FUNCTION_BLOCK TaskCenterMSGParse (* Service Interface Function Block Type *)
  (* Standard: 61499-2 *)
  (* Version 0.0, 2018-06-21, 4DIAC-IDE, 4DIAC-Consortium *)
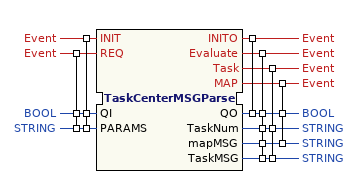
  EVENT_INPUT
    INIT WITH QI, PARAMS; (* Service Initialization *)
    REQ WITH QI, PARAMS; (* Service Request *)
  END_EVENT
  EVENT_OUTPUT
    INITO WITH QO; (* Initialization Confirm *)
    Evaluate WITH QO, TaskMSG, TaskNum, mapMSG; (* Indication from Resource *)
    Task WITH TaskMSG, TaskNum;
    MAP WITH QO, mapMSG;
  END_EVENT
  VAR_INPUT
    QI : BOOL; (* Event Input Qualifier *)
    PARAMS : STRING; (* Service Parameters *)
  END_VAR
  VAR_OUTPUT
    QO : BOOL; (* Event Output Qualifier *)
    TaskNum : STRING;
    mapMSG : STRING; (* MAP msg *)
    TaskMSG : STRING; (* Input data from resource *)
  END_VAR
  SERVICE APPLICATION/RESOURCE (* Service Interface Function Block Type *)
    SEQUENCE normal_establishment
      APPLICATION.INIT+(PARAMS) -> RESOURCE.initialize(PARAMS) -> APPLICATION.INITO+();
    END_SEQUENCE
    SEQUENCE unsuccessful_establishment
      APPLICATION.INIT+(PARAMS) -> RESOURCE.initialize(PARAMS) -> APPLICATION.INITO-(STATUS);
    END_SEQUENCE
    SEQUENCE request_confirm
      APPLICATION.REQ+(SD) -> RESOURCE.request(SD) -> APPLICATION.CNF+(RD);
    END_SEQUENCE
    SEQUENCE request_inhibited
      APPLICATION.REQ-(SD) -> APPLICATION.CNF-(STATUS);
    END_SEQUENCE
    SEQUENCE request_error
      APPLICATION.REQ+(SD) -> RESOURCE.request(SD) -> APPLICATION.CNF-(STATUS);
    END_SEQUENCE
    SEQUENCE indication_response
      RESOURCE.indicate(RD) -> APPLICATION.IND+(RD);
      APPLICATION.RSP(QI,SD) -> RESOURCE.response(QI,SD);
    END_SEQUENCE
    SEQUENCE indication_inhibited
      RESOURCE.indicate(RD,QI=FALSE) -> RESOURCE.inhibited();
    END_SEQUENCE
    SEQUENCE error_indication
      RESOURCE.error(STATUS) -> APPLICATION.IND-(STATUS);
    END_SEQUENCE
    SEQUENCE application_initiated_termination
      APPLICATION.INIT-() -> RESOURCE.terminate() -> APPLICATION.INITO-(STATUS);
    END_SEQUENCE
    SEQUENCE resource_initiated_termination
      -> APPLICATION.INITO-(STATUS);
    END_SEQUENCE
  END_SERVICE
END_FUNCTION_BLOCK
